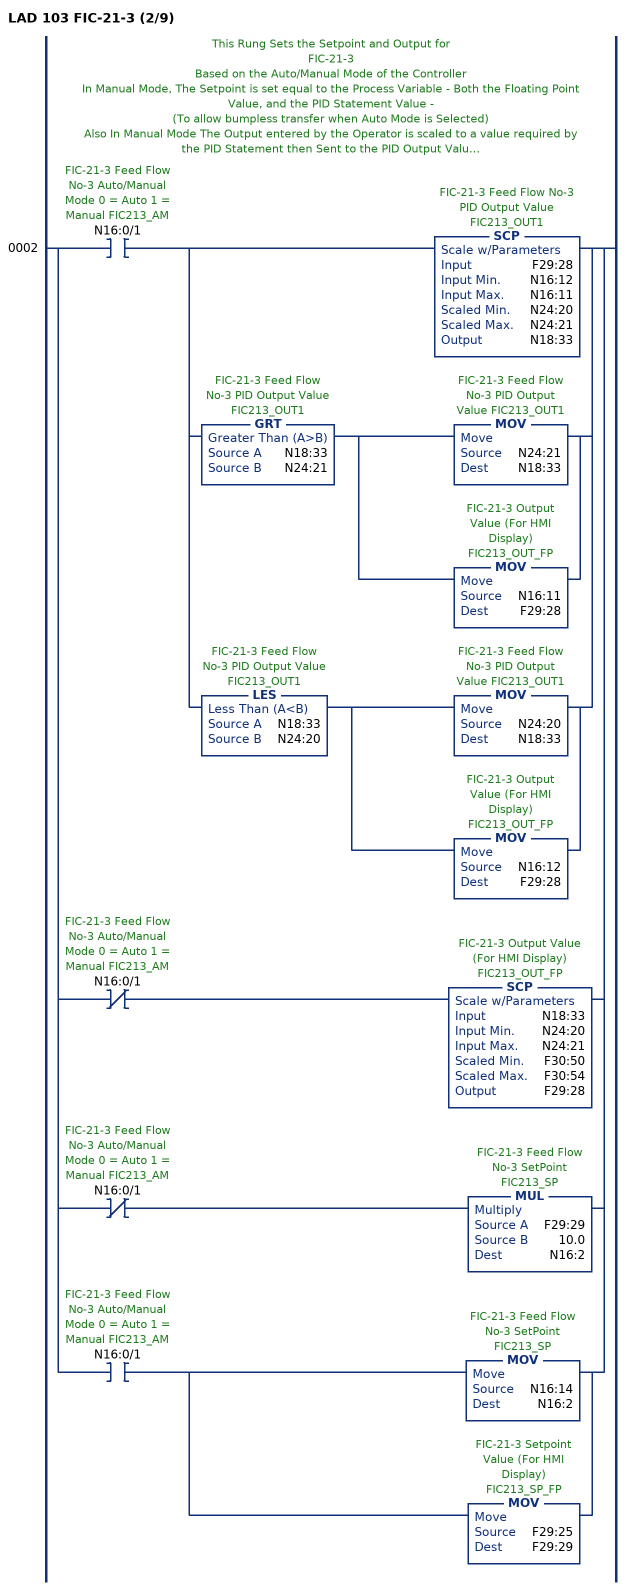
% Rung: 2 %
% This Rung Sets the Setpoint and Output for
% FIC-21-3
% Based on the Auto/Manual Mode of the Controller
% In Manual Mode, The Setpoint is set equal to the Process Variable - Both the Floating Point Value, and the PID Statement Value -
% (To allow bumpless transfer when Auto Mode is Selected)
% Also In Manual Mode The Output entered by the Operator is scaled to a value required by the PID Statement then Sent to the PID Output Value
% 
% In Auto Mode, The Setpoint is Entered by the Operator from Any HMI terminal, Multiplied by 10, and placed in the PID Statement's Setpoint Location
% Also In Auto Mode, the Output (used by the Operator) is set equal to the actual value of the pID statement
% (To allow bumpless transfer when Manual Mode is Selected) %
SOR BST XIC N16:0/1 BST SCP F29:28 N16:12 N16:11 N24:20 N24:21 N18:33 NXB GRT N18:33 N24:21 BST MOV N24:21 N18:33 NXB MOV N16:11 F29:28 BND NXB LES N18:33 N24:20 BST MOV N24:20 N18:33 NXB MOV N16:12 F29:28 BND BND NXB XIO N16:0/1 SCP N18:33 N24:20 N24:21 F30:50 F30:54 F29:28 NXB XIO N16:0/1 MUL F29:29 10.0 N16:2 NXB XIC N16:0/1 BST MOV N16:14 N16:2 NXB MOV F29:25 F29:29 BND BND EOR
%   N16:0/1  FIC213_AM  "FIC-21-3 Feed Flow No-3 Auto/Manual Mode 0 = Auto 1 = Manual" %
%   F29:28  FIC213_OUT_FP  "FIC-21-3 Output Value (For HMI Display)" %
%   N16:12  FIC213_OMIN  "FIC-21-3 Feed Flow No-3 Output Minimum" %
%   N16:11  FIC213_OMAX  "FIC-21-3 Feed Flow No-3 Output Maximum" %
%   N24:20  PID_MIN  "PID Statement Minimum Value" %
%   N24:21  PID_MAX  "PID Statement Maximum Value" %
%   N18:33  FIC213_OUT1  "FIC-21-3 Feed Flow No-3 PID Output Value" %
%   F30:50  SIC213_MIN  "SIC-21-3 PU-21-3 Feed Pump No-3 Speed 0% Value (For HMI Display)" %
%   F30:54  SIC213_MAX  "SIC-21-3 PU-21-3 Feed Pump No-3 Freq at 100% Value (For HMI Display)" %
%   F29:29  FIC213_SP_FP  "FIC-21-3 Setpoint Value (For HMI Display)" %
%   N16:2  FIC213_SP  "FIC-21-3 Feed Flow No-3 SetPoint" %
%   N16:14  FIC213_PV  "FIC-21-3 Feed Flow No-3 Scaled Process Variable" %
%   F29:25  FIC213_PV_FP  "FIC-21-3 PV Value (For HMI Display)" %

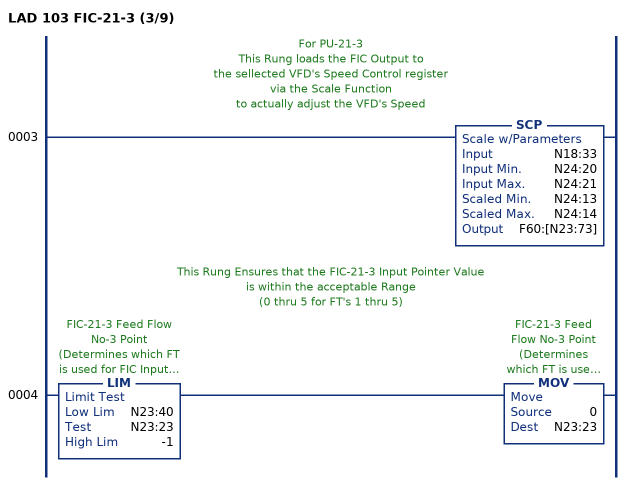
% Rung: 3 %
% For PU-21-3
% This Rung loads the FIC Output to
% the sellected VFD's Speed Control register
% via the Scale Function
% to actually adjust the VFD's Speed %
SOR SCP N18:33 N24:20 N24:21 N24:13 N24:14 F60:[N23:73] EOR
%   N18:33  FIC213_OUT1  "FIC-21-3 Feed Flow No-3 PID Output Value" %
%   N24:20  PID_MIN  "PID Statement Minimum Value" %
%   N24:21  PID_MAX  "PID Statement Maximum Value" %
%   N24:13  AO_MIN_OE4  "Analog Output Minimum Value Generates 4 mA DC (To OE4 AO Module)" %
%   N24:14  AO_MAX_OE4  "Analog Output Maximum Value Generates 20 mA DC (To OE4 AO Module)" %
%   N23:73  FIC213_OUT_PTR  "FIC-21-3 Feed Flow No-3 Output Pointer Determines which VFD is controled by FIC" %
% Rung: 4 %
% This Rung Ensures that the FIC-21-3 Input Pointer Value
% is within the acceptable Range
% (0 thru 5 for FT's 1 thru 5) %
SOR LIM N23:40 N23:23 -1 MOV 0 N23:23 EOR
%   N23:40  MAX_FT_ALLOWED_1  "Maximum Number of FTs Available Plus 1" %
%   N23:23  FIC213_IN_PTR  "FIC-21-3 Feed Flow No-3 Point (Determines which FT is used for FIC Input)" %

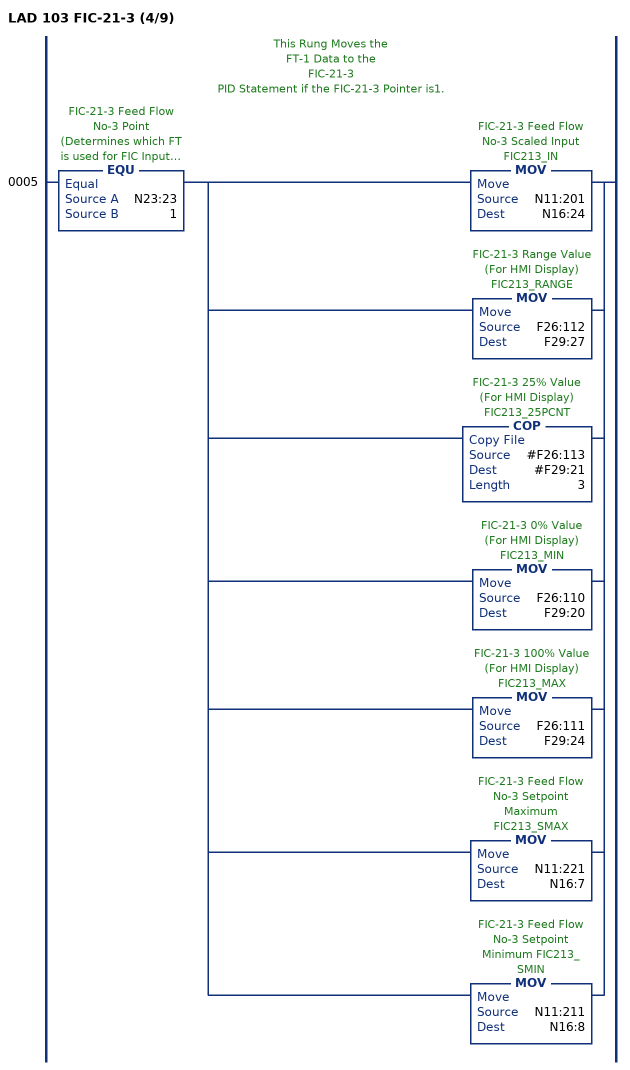
% Rung: 5 %
% This Rung Moves the
% FT-1 Data to the
% FIC-21-3
% PID Statement if the FIC-21-3 Pointer is1. %
SOR EQU N23:23 1 BST MOV N11:201 N16:24 NXB MOV F26:112 F29:27 NXB COP #F26:113 #F29:21 3 NXB MOV F26:110 F29:20 NXB MOV F26:111 F29:24 NXB MOV N11:221 N16:7 NXB MOV N11:211 N16:8 BND EOR
%   N23:23  FIC213_IN_PTR  "FIC-21-3 Feed Flow No-3 Point (Determines which FT is used for FIC Input)" %
%   N11:201  FT01_PID_IN  "FT-1 Flow Transmitter No-1 PID Statement Input Value" %
%   N16:24  FIC213_IN  "FIC-21-3 Feed Flow No-3 Scaled Input" %
%   F26:112  FT01_RANGE  "FT-1 Range Value (Max-Min)" %
%   F29:27  FIC213_RANGE  "FIC-21-3 Range Value (For HMI Display)" %
%   F26:113  FT01_25PCNT_VALUE  "FT-1 25% Range Value For HMI Display" %
%   F29:21  FIC213_25PCNT  "FIC-21-3 25% Value (For HMI Display)" %
%   F26:110  FT01_MIN  "FT-1 Minimum Value" %
%   F29:20  FIC213_MIN  "FIC-21-3 0% Value (For HMI Display)" %
%   F26:111  FT01_MAX  "FT-1 Maximum Value" %
%   F29:24  FIC213_MAX  "FIC-21-3 100% Value (For HMI Display)" %
%   N11:221  FT01_PID_MAX  "FT-1 Flow Transmitter No-1 PID Statement Maximum Input Value" %
%   N16:7  FIC213_SMAX  "FIC-21-3 Feed Flow No-3 Setpoint Maximum" %
%   N11:211  FT01_PID_MIN  "FT-1 Flow Transmitter No-1 PID Statement Minimum Input Value" %
%   N16:8  FIC213_SMIN  "FIC-21-3 Feed Flow No-3 Setpoint Minimum" %

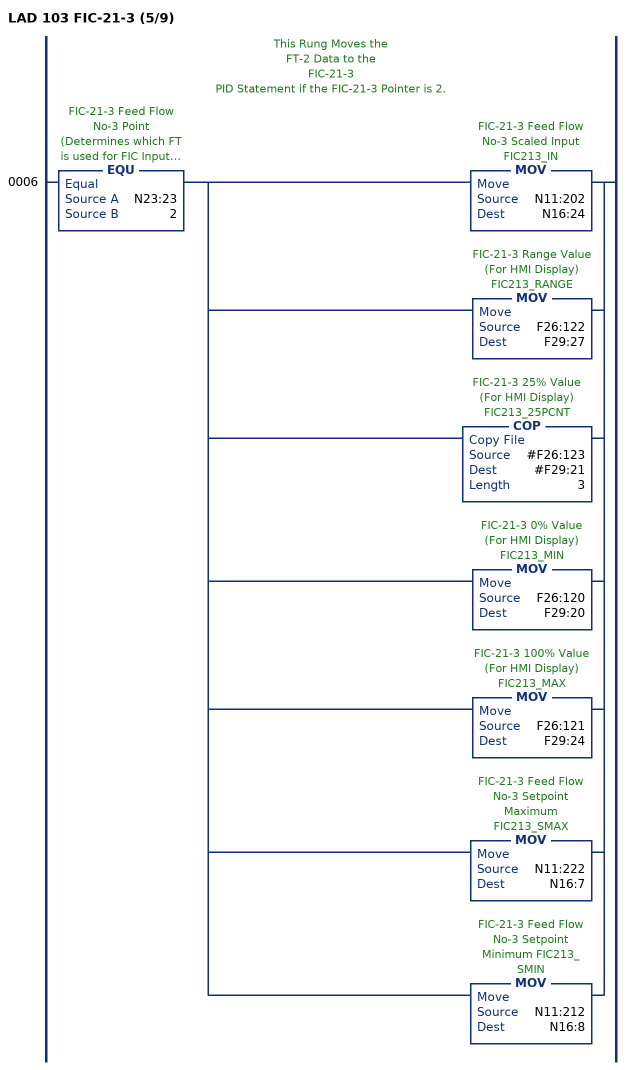
% Rung: 6 %
% This Rung Moves the
% FT-2 Data to the
% FIC-21-3
% PID Statement if the FIC-21-3 Pointer is 2. %
SOR EQU N23:23 2 BST MOV N11:202 N16:24 NXB MOV F26:122 F29:27 NXB COP #F26:123 #F29:21 3 NXB MOV F26:120 F29:20 NXB MOV F26:121 F29:24 NXB MOV N11:222 N16:7 NXB MOV N11:212 N16:8 BND EOR
%   N23:23  FIC213_IN_PTR  "FIC-21-3 Feed Flow No-3 Point (Determines which FT is used for FIC Input)" %
%   N11:202  FT02_PID_IN  "FT-2 Flow Transmitter No-2 PID Statement Input Value" %
%   N16:24  FIC213_IN  "FIC-21-3 Feed Flow No-3 Scaled Input" %
%   F26:122  FT02_RANGE  "FT-2 Range Value (Max-Min)" %
%   F29:27  FIC213_RANGE  "FIC-21-3 Range Value (For HMI Display)" %
%   F26:123  FT02_25PCNT_VALUE  "FT-2 25% Range Value For HMI Display" %
%   F29:21  FIC213_25PCNT  "FIC-21-3 25% Value (For HMI Display)" %
%   F26:120  FT02_MIN  "FT-2 Minimum Value" %
%   F29:20  FIC213_MIN  "FIC-21-3 0% Value (For HMI Display)" %
%   F26:121  FT02_MAX  "FT-2 Maximum Value" %
%   F29:24  FIC213_MAX  "FIC-21-3 100% Value (For HMI Display)" %
%   N11:222  FT02_PID_MAX  "FT-2 Flow Transmitter No-2 PID Statement Maximum Input Value" %
%   N16:7  FIC213_SMAX  "FIC-21-3 Feed Flow No-3 Setpoint Maximum" %
%   N11:212  FT02_PID_MIN  "FT-2 Flow Transmitter No-2 PID Statement Minimum Input Value" %
%   N16:8  FIC213_SMIN  "FIC-21-3 Feed Flow No-3 Setpoint Minimum" %

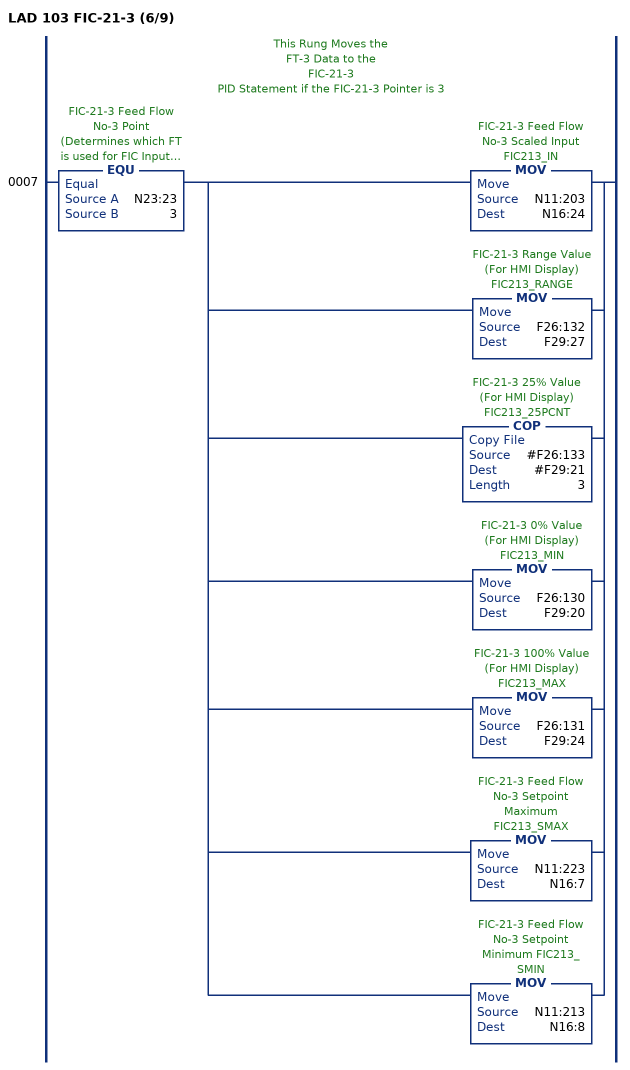
% Rung: 7 %
% This Rung Moves the
% FT-3 Data to the
% FIC-21-3
% PID Statement if the FIC-21-3 Pointer is 3 %
SOR EQU N23:23 3 BST MOV N11:203 N16:24 NXB MOV F26:132 F29:27 NXB COP #F26:133 #F29:21 3 NXB MOV F26:130 F29:20 NXB MOV F26:131 F29:24 NXB MOV N11:223 N16:7 NXB MOV N11:213 N16:8 BND EOR
%   N23:23  FIC213_IN_PTR  "FIC-21-3 Feed Flow No-3 Point (Determines which FT is used for FIC Input)" %
%   N11:203  FT03_PID_IN  "FT-3 Flow Transmitter No-3 PID Statement Input Value" %
%   N16:24  FIC213_IN  "FIC-21-3 Feed Flow No-3 Scaled Input" %
%   F26:132  FT03_RANGE  "FT-3 Range Value (Max-Min)" %
%   F29:27  FIC213_RANGE  "FIC-21-3 Range Value (For HMI Display)" %
%   F26:133  FT03_25PCNT_VALUE  "FT-3 25% Range Value For HMI Display" %
%   F29:21  FIC213_25PCNT  "FIC-21-3 25% Value (For HMI Display)" %
%   F26:130  FT03_MIN  "FT-3 Minimum Value" %
%   F29:20  FIC213_MIN  "FIC-21-3 0% Value (For HMI Display)" %
%   F26:131  FT03_MAX  "FT-3 Maximum Value" %
%   F29:24  FIC213_MAX  "FIC-21-3 100% Value (For HMI Display)" %
%   N11:223  FT03_PID_MAX  "FT-3 Flow Transmitter No-3 PID Statement Maximum Input Value" %
%   N16:7  FIC213_SMAX  "FIC-21-3 Feed Flow No-3 Setpoint Maximum" %
%   N11:213  FT03_PID_MIN  "FT-3 Flow Transmitter No-3 PID Statement Minimum Input Value" %
%   N16:8  FIC213_SMIN  "FIC-21-3 Feed Flow No-3 Setpoint Minimum" %

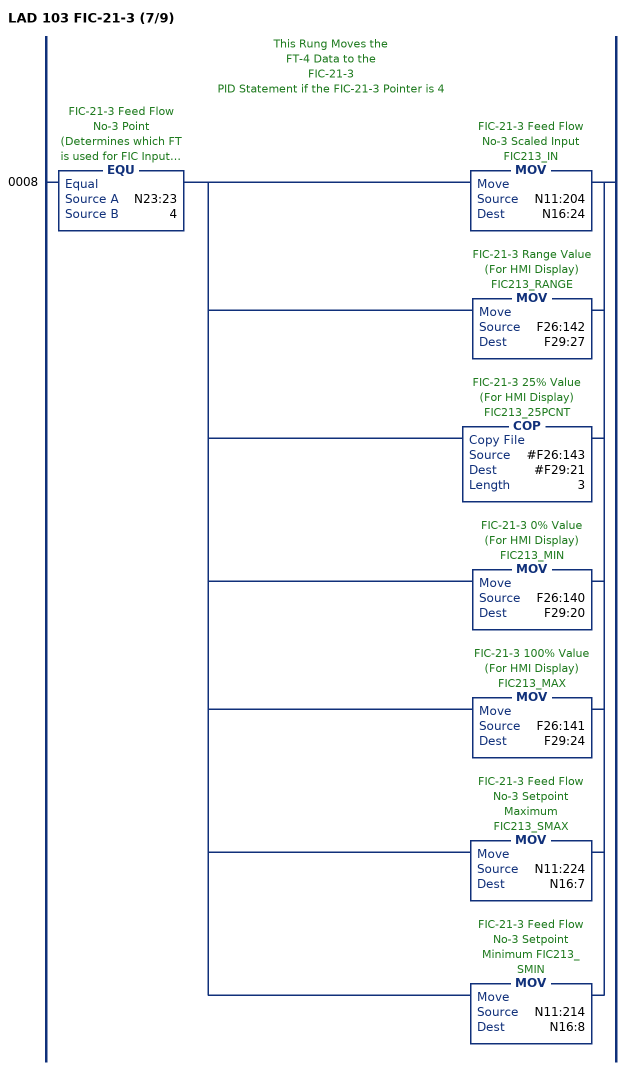
% Rung: 8 %
% This Rung Moves the
% FT-4 Data to the
% FIC-21-3
% PID Statement if the FIC-21-3 Pointer is 4 %
SOR EQU N23:23 4 BST MOV N11:204 N16:24 NXB MOV F26:142 F29:27 NXB COP #F26:143 #F29:21 3 NXB MOV F26:140 F29:20 NXB MOV F26:141 F29:24 NXB MOV N11:224 N16:7 NXB MOV N11:214 N16:8 BND EOR
%   N23:23  FIC213_IN_PTR  "FIC-21-3 Feed Flow No-3 Point (Determines which FT is used for FIC Input)" %
%   N11:204  FT04_PID_IN  "FT-4 Flow Transmitter No-4 PID Statement Input Value" %
%   N16:24  FIC213_IN  "FIC-21-3 Feed Flow No-3 Scaled Input" %
%   F26:142  FT04_RANGE  "FT-4 Range Value (Max-Min)" %
%   F29:27  FIC213_RANGE  "FIC-21-3 Range Value (For HMI Display)" %
%   F26:143  FT04_25PCNT_VALUE  "FT-4 25% Range Value For HMI Display" %
%   F29:21  FIC213_25PCNT  "FIC-21-3 25% Value (For HMI Display)" %
%   F26:140  FT04_MIN  "FT-4 Minimum Value" %
%   F29:20  FIC213_MIN  "FIC-21-3 0% Value (For HMI Display)" %
%   F26:141  FT04_MAX  "FT-4 Maximum Value" %
%   F29:24  FIC213_MAX  "FIC-21-3 100% Value (For HMI Display)" %
%   N11:224  FT04_PID_MAX  "FT-4 Flow Transmitter No-4 PID Statement Maximum Input Value" %
%   N16:7  FIC213_SMAX  "FIC-21-3 Feed Flow No-3 Setpoint Maximum" %
%   N11:214  FT04_PID_MIN  "FT-4 Flow Transmitter No-4 PID Statement Minimum Input Value" %
%   N16:8  FIC213_SMIN  "FIC-21-3 Feed Flow No-3 Setpoint Minimum" %

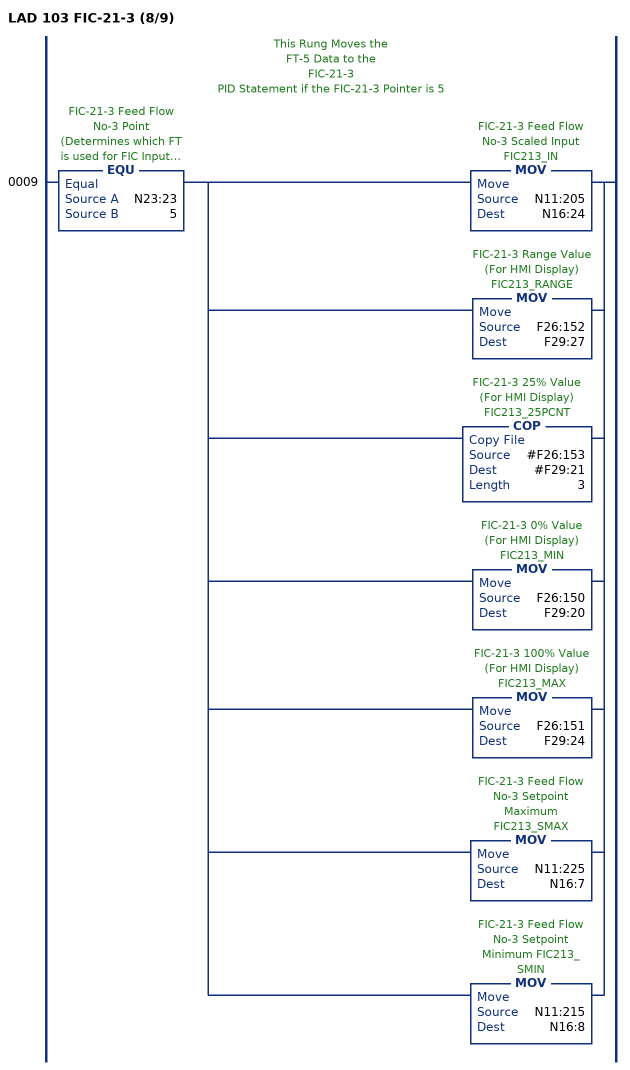
% Rung: 9 %
% This Rung Moves the
% FT-5 Data to the
% FIC-21-3
%  PID Statement if the FIC-21-3 Pointer is 5 %
SOR EQU N23:23 5 BST MOV N11:205 N16:24 NXB MOV F26:152 F29:27 NXB COP #F26:153 #F29:21 3 NXB MOV F26:150 F29:20 NXB MOV F26:151 F29:24 NXB MOV N11:225 N16:7 NXB MOV N11:215 N16:8 BND EOR
%   N23:23  FIC213_IN_PTR  "FIC-21-3 Feed Flow No-3 Point (Determines which FT is used for FIC Input)" %
%   N11:205  FT05_PID_IN  "FT-5 Flow Transmitter No-5 PID Statement Input Value" %
%   N16:24  FIC213_IN  "FIC-21-3 Feed Flow No-3 Scaled Input" %
%   F26:152  FT05_RANGE  "FT-5 Range Value (Max-Min)" %
%   F29:27  FIC213_RANGE  "FIC-21-3 Range Value (For HMI Display)" %
%   F26:153  FT05_25PCNT_VALUE  "FT-5 25% Range Value For HMI Display" %
%   F29:21  FIC213_25PCNT  "FIC-21-3 25% Value (For HMI Display)" %
%   F26:150  FT05_MIN  "FT-5 Minimum Value" %
%   F29:20  FIC213_MIN  "FIC-21-3 0% Value (For HMI Display)" %
%   F26:151  FT05_MAX  "FT-5 Maximum Value" %
%   F29:24  FIC213_MAX  "FIC-21-3 100% Value (For HMI Display)" %
%   N11:225  FT05_PID_MAX  "FT-5 Flow Transmitter No-5 PID Statement Maximum Input Value" %
%   N16:7  FIC213_SMAX  "FIC-21-3 Feed Flow No-3 Setpoint Maximum" %
%   N11:215  FT05_PID_MIN  "FT-5 Flow Transmitter No-5 PID Statement Minimum Input Value" %
%   N16:8  FIC213_SMIN  "FIC-21-3 Feed Flow No-3 Setpoint Minimum" %

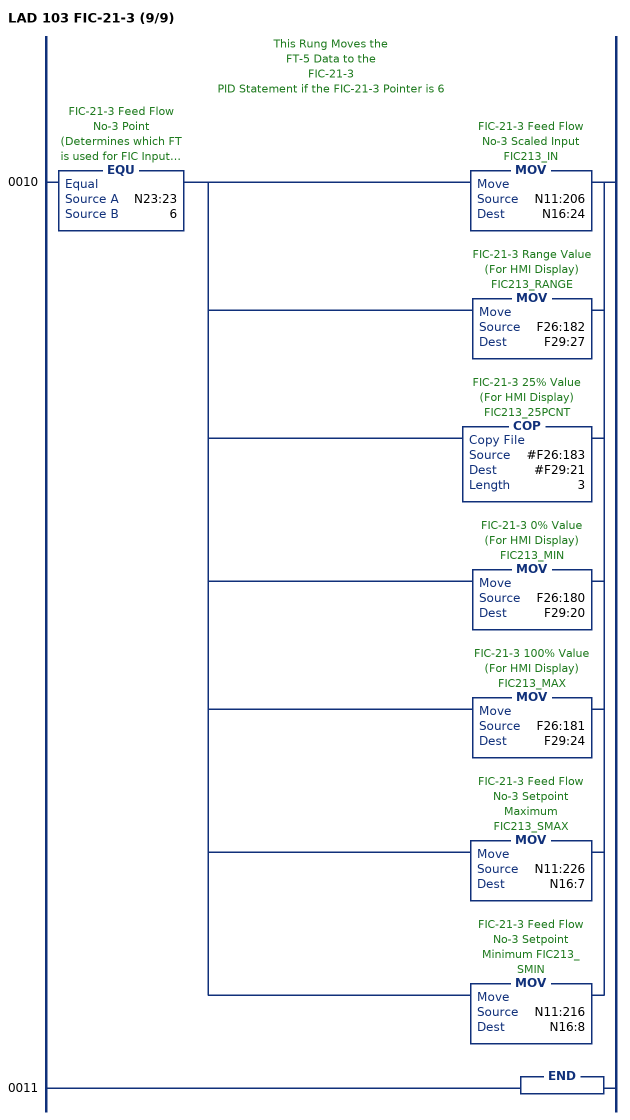
% Rung: 10 %
% This Rung Moves the
% FT-5 Data to the
% FIC-21-3
%  PID Statement if the FIC-21-3 Pointer is 6 %
SOR EQU N23:23 6 BST MOV N11:206 N16:24 NXB MOV F26:182 F29:27 NXB COP #F26:183 #F29:21 3 NXB MOV F26:180 F29:20 NXB MOV F26:181 F29:24 NXB MOV N11:226 N16:7 NXB MOV N11:216 N16:8 BND EOR
%   N23:23  FIC213_IN_PTR  "FIC-21-3 Feed Flow No-3 Point (Determines which FT is used for FIC Input)" %
%   N11:206  FT06_PID_IN  "FT-6 Flow Transmitter No-6 PID Statement Input Value" %
%   N16:24  FIC213_IN  "FIC-21-3 Feed Flow No-3 Scaled Input" %
%   F26:182  FT06_RANGE  "FT-6 Range Value (Max-Min)" %
%   F29:27  FIC213_RANGE  "FIC-21-3 Range Value (For HMI Display)" %
%   F26:183  FT06_25PCNT_VALUE  "FT-6 25% Range Value For HMI Display" %
%   F29:21  FIC213_25PCNT  "FIC-21-3 25% Value (For HMI Display)" %
%   F26:180  FT06_MIN  "FT-6 Minimum Value" %
%   F29:20  FIC213_MIN  "FIC-21-3 0% Value (For HMI Display)" %
%   F26:181  FT06_MAX  "FT-6 Maximum Value" %
%   F29:24  FIC213_MAX  "FIC-21-3 100% Value (For HMI Display)" %
%   N11:226  FT06_PID_MAX  "FT-6 Flow Transmitter No-6 PID Statement Maximum Input Value" %
%   N16:7  FIC213_SMAX  "FIC-21-3 Feed Flow No-3 Setpoint Maximum" %
%   N11:216  FT06_PID_MIN  "FT-6 Flow Transmitter No-6 PID Statement Minimum Input Value" %
%   N16:8  FIC213_SMIN  "FIC-21-3 Feed Flow No-3 Setpoint Minimum" %
% Rung: 11 %
SOR END EOR

LADDER 104 "FIC-21-4"    % Feed Flow No-4 PID Controls %
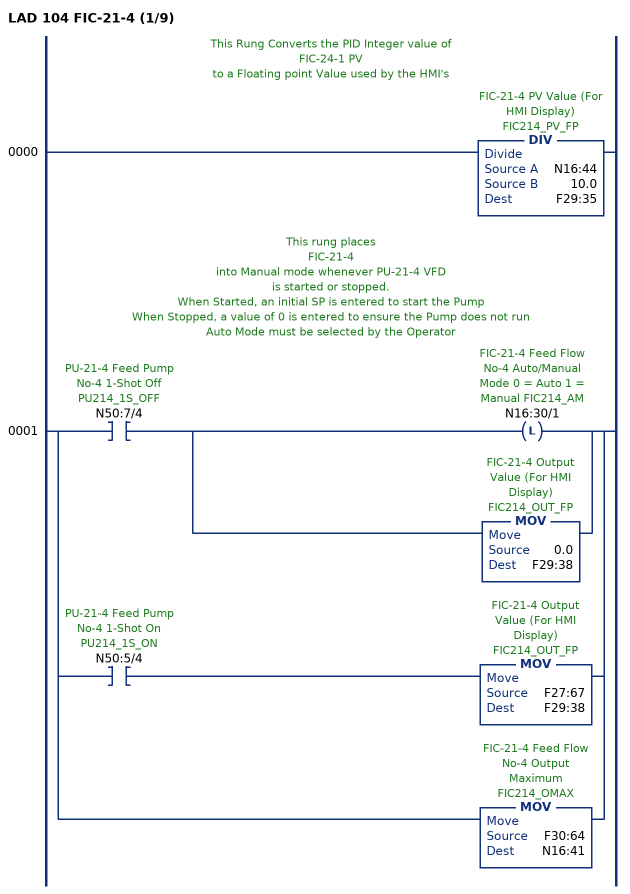
% Rung: 0 %
% This Rung Converts the PID Integer value of
% FIC-24-1 PV
% to a Floating point Value used by the HMI's %
SOR DIV N16:44 10.0 F29:35 EOR
%   N16:44  FIC214_PV  "FIC-21-4 Feed Flow No-4 Scaled Process Variable" %
%   F29:35  FIC214_PV_FP  "FIC-21-4 PV Value (For HMI Display)" %
% Rung: 1 %
% This rung places
% FIC-21-4
% into Manual mode whenever PU-21-4 VFD
% is started or stopped.
% When Started, an initial SP is entered to start the Pump
% When Stopped, a value of 0 is entered to ensure the Pump does not run
% Auto Mode must be selected by the Operator %
SOR BST XIC N50:7/4 BST OTL N16:30/1 NXB MOV 0.0 F29:38 BND NXB XIC N50:5/4 MOV F27:67 F29:38 NXB MOV F30:64 N16:41 BND EOR
%   N50:7/4  PU214_1S_OFF  "PU-21-4 Feed Pump No-4 1-Shot Off" %
%   N16:30/1  FIC214_AM  "FIC-21-4 Feed Flow No-4 Auto/Manual Mode 0 = Auto 1 = Manual" %
%   F29:38  FIC214_OUT_FP  "FIC-21-4 Output Value (For HMI Display)" %
%   N50:5/4  PU214_1S_ON  "PU-21-4 Feed Pump No-4 1-Shot On" %
%   F27:67  SIC214_INIT_SP  "SIC-21-4 Initial Speed Setpoint (Hz)" %
%   F30:64  SIC214_MAX  "SIC-21-4 PU-21-4 Feed Pump No-4 Freq at 100% Value (For HMI Display)" %
%   N16:41  FIC214_OMAX  "FIC-21-4 Feed Flow No-4 Output Maximum" %

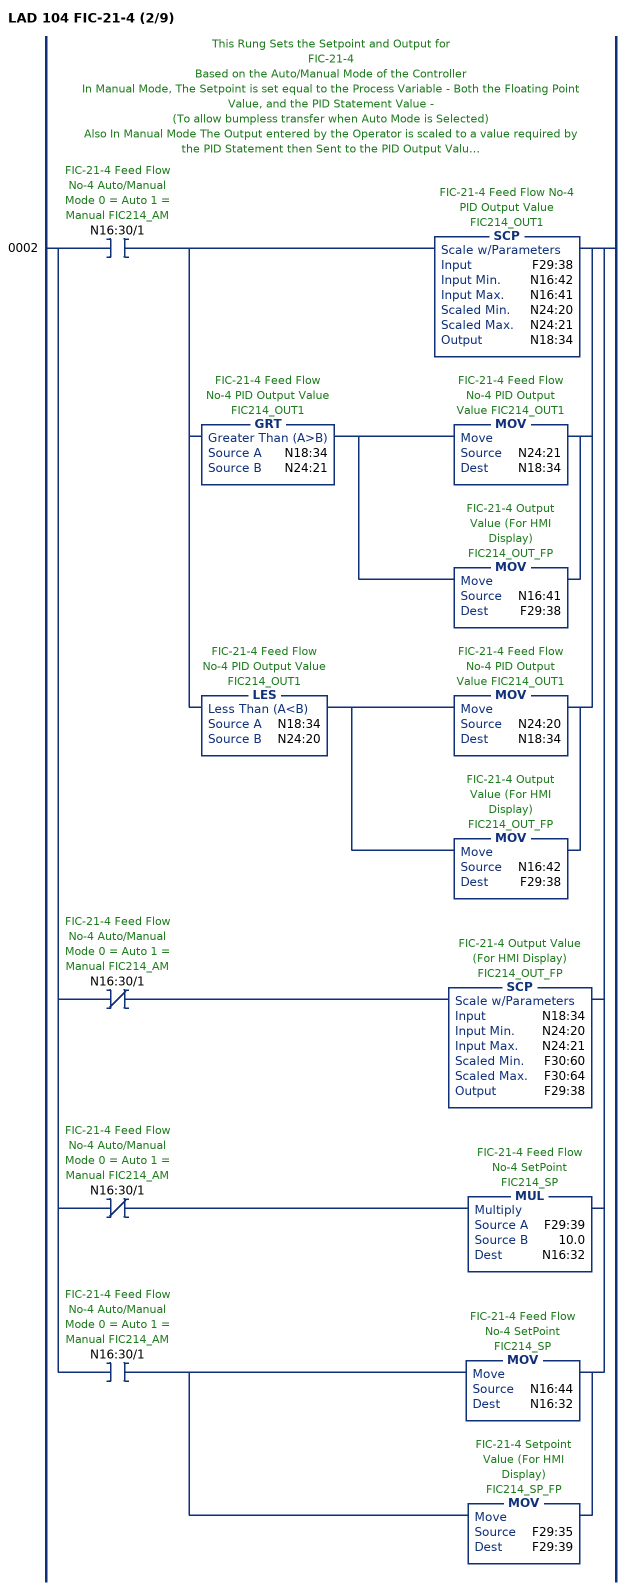
% Rung: 2 %
% This Rung Sets the Setpoint and Output for
% FIC-21-4
% Based on the Auto/Manual Mode of the Controller
% In Manual Mode, The Setpoint is set equal to the Process Variable - Both the Floating Point Value, and the PID Statement Value -
% (To allow bumpless transfer when Auto Mode is Selected)
% Also In Manual Mode The Output entered by the Operator is scaled to a value required by the PID Statement then Sent to the PID Output Value
% 
% In Auto Mode, The Setpoint is Entered by the Operator from Any HMI terminal, Multiplied by 10, and placed in the PID Statement's Setpoint Location
% Also In Auto Mode, the Output (used by the Operator) is set equal to the actual value of the pID statement
% (To allow bumpless transfer when Manual Mode is Selected) %
SOR BST XIC N16:30/1 BST SCP F29:38 N16:42 N16:41 N24:20 N24:21 N18:34 NXB GRT N18:34 N24:21 BST MOV N24:21 N18:34 NXB MOV N16:41 F29:38 BND NXB LES N18:34 N24:20 BST MOV N24:20 N18:34 NXB MOV N16:42 F29:38 BND BND NXB XIO N16:30/1 SCP N18:34 N24:20 N24:21 F30:60 F30:64 F29:38 NXB XIO N16:30/1 MUL F29:39 10.0 N16:32 NXB XIC N16:30/1 BST MOV N16:44 N16:32 NXB MOV F29:35 F29:39 BND BND EOR
%   N16:30/1  FIC214_AM  "FIC-21-4 Feed Flow No-4 Auto/Manual Mode 0 = Auto 1 = Manual" %
%   F29:38  FIC214_OUT_FP  "FIC-21-4 Output Value (For HMI Display)" %
%   N16:42  FIC214_OMIN  "FIC-21-4 Feed Flow No-4 Output Minimum" %
%   N16:41  FIC214_OMAX  "FIC-21-4 Feed Flow No-4 Output Maximum" %
%   N24:20  PID_MIN  "PID Statement Minimum Value" %
%   N24:21  PID_MAX  "PID Statement Maximum Value" %
%   N18:34  FIC214_OUT1  "FIC-21-4 Feed Flow No-4 PID Output Value" %
%   F30:60  SIC214_MIN  "SIC-21-4 PU-21-4 Feed Pump No-4 Speed 0% Value (For HMI Display)" %
%   F30:64  SIC214_MAX  "SIC-21-4 PU-21-4 Feed Pump No-4 Freq at 100% Value (For HMI Display)" %
%   F29:39  FIC214_SP_FP  "FIC-21-4 Setpoint Value (For HMI Display)" %
%   N16:32  FIC214_SP  "FIC-21-4 Feed Flow No-4 SetPoint" %
%   N16:44  FIC214_PV  "FIC-21-4 Feed Flow No-4 Scaled Process Variable" %
%   F29:35  FIC214_PV_FP  "FIC-21-4 PV Value (For HMI Display)" %

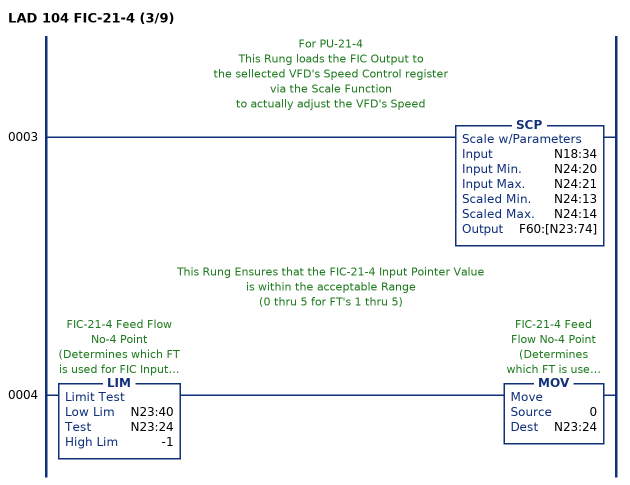
% Rung: 3 %
% For PU-21-4
% This Rung loads the FIC Output to
% the sellected VFD's Speed Control register
% via the Scale Function
% to actually adjust the VFD's Speed %
SOR SCP N18:34 N24:20 N24:21 N24:13 N24:14 F60:[N23:74] EOR
%   N18:34  FIC214_OUT1  "FIC-21-4 Feed Flow No-4 PID Output Value" %
%   N24:20  PID_MIN  "PID Statement Minimum Value" %
%   N24:21  PID_MAX  "PID Statement Maximum Value" %
%   N24:13  AO_MIN_OE4  "Analog Output Minimum Value Generates 4 mA DC (To OE4 AO Module)" %
%   N24:14  AO_MAX_OE4  "Analog Output Maximum Value Generates 20 mA DC (To OE4 AO Module)" %
%   N23:74  FIC214_OUT_PTR  "FIC-21-4 Feed Flow No-4 Output Pointer Determines which VFD is controled by FIC" %
% Rung: 4 %
% This Rung Ensures that the FIC-21-4 Input Pointer Value
% is within the acceptable Range
% (0 thru 5 for FT's 1 thru 5) %
SOR LIM N23:40 N23:24 -1 MOV 0 N23:24 EOR
%   N23:40  MAX_FT_ALLOWED_1  "Maximum Number of FTs Available Plus 1" %
%   N23:24  FIC214_IN_PTR  "FIC-21-4 Feed Flow No-4 Point (Determines which FT is used for FIC Input)" %

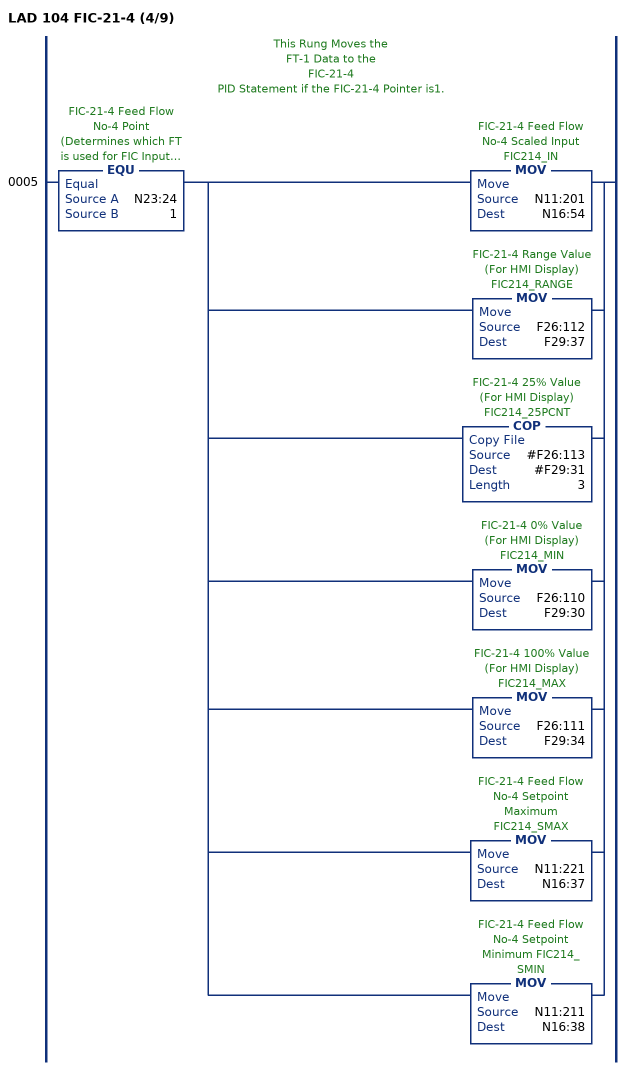
% Rung: 5 %
% This Rung Moves the
% FT-1 Data to the
% FIC-21-4
% PID Statement if the FIC-21-4 Pointer is1. %
SOR EQU N23:24 1 BST MOV N11:201 N16:54 NXB MOV F26:112 F29:37 NXB COP #F26:113 #F29:31 3 NXB MOV F26:110 F29:30 NXB MOV F26:111 F29:34 NXB MOV N11:221 N16:37 NXB MOV N11:211 N16:38 BND EOR
%   N23:24  FIC214_IN_PTR  "FIC-21-4 Feed Flow No-4 Point (Determines which FT is used for FIC Input)" %
%   N11:201  FT01_PID_IN  "FT-1 Flow Transmitter No-1 PID Statement Input Value" %
%   N16:54  FIC214_IN  "FIC-21-4 Feed Flow No-4 Scaled Input" %
%   F26:112  FT01_RANGE  "FT-1 Range Value (Max-Min)" %
%   F29:37  FIC214_RANGE  "FIC-21-4 Range Value (For HMI Display)" %
%   F26:113  FT01_25PCNT_VALUE  "FT-1 25% Range Value For HMI Display" %
%   F29:31  FIC214_25PCNT  "FIC-21-4 25% Value (For HMI Display)" %
%   F26:110  FT01_MIN  "FT-1 Minimum Value" %
%   F29:30  FIC214_MIN  "FIC-21-4 0% Value (For HMI Display)" %
%   F26:111  FT01_MAX  "FT-1 Maximum Value" %
%   F29:34  FIC214_MAX  "FIC-21-4 100% Value (For HMI Display)" %
%   N11:221  FT01_PID_MAX  "FT-1 Flow Transmitter No-1 PID Statement Maximum Input Value" %
%   N16:37  FIC214_SMAX  "FIC-21-4 Feed Flow No-4 Setpoint Maximum" %
%   N11:211  FT01_PID_MIN  "FT-1 Flow Transmitter No-1 PID Statement Minimum Input Value" %
%   N16:38  FIC214_SMIN  "FIC-21-4 Feed Flow No-4 Setpoint Minimum" %

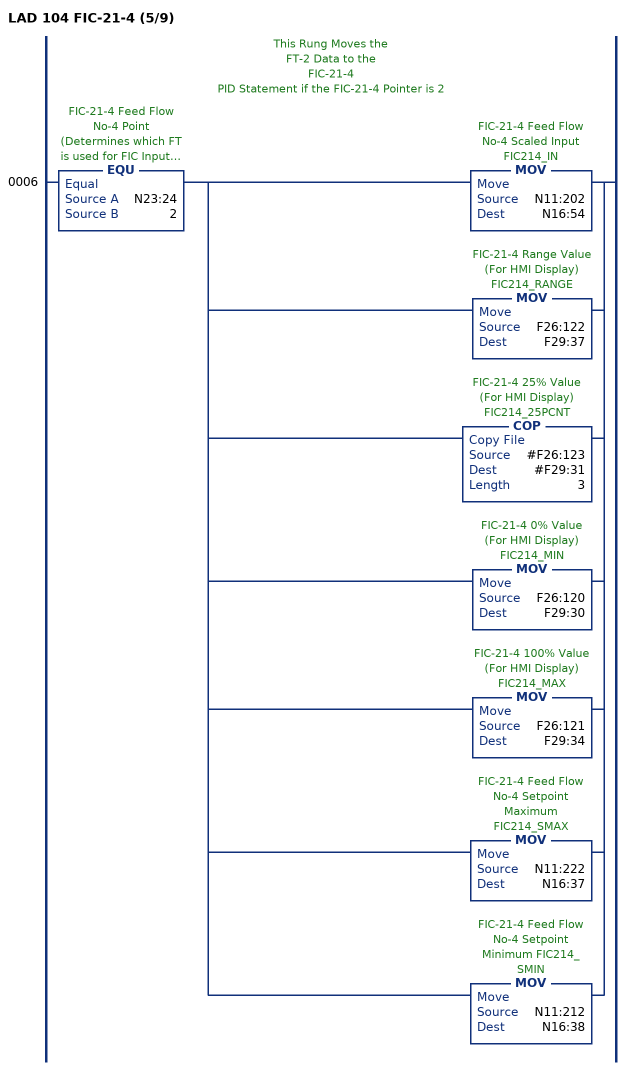
% Rung: 6 %
% This Rung Moves the
% FT-2 Data to the
% FIC-21-4
% PID Statement if the FIC-21-4 Pointer is 2 %
SOR EQU N23:24 2 BST MOV N11:202 N16:54 NXB MOV F26:122 F29:37 NXB COP #F26:123 #F29:31 3 NXB MOV F26:120 F29:30 NXB MOV F26:121 F29:34 NXB MOV N11:222 N16:37 NXB MOV N11:212 N16:38 BND EOR
%   N23:24  FIC214_IN_PTR  "FIC-21-4 Feed Flow No-4 Point (Determines which FT is used for FIC Input)" %
%   N11:202  FT02_PID_IN  "FT-2 Flow Transmitter No-2 PID Statement Input Value" %
%   N16:54  FIC214_IN  "FIC-21-4 Feed Flow No-4 Scaled Input" %
%   F26:122  FT02_RANGE  "FT-2 Range Value (Max-Min)" %
%   F29:37  FIC214_RANGE  "FIC-21-4 Range Value (For HMI Display)" %
%   F26:123  FT02_25PCNT_VALUE  "FT-2 25% Range Value For HMI Display" %
%   F29:31  FIC214_25PCNT  "FIC-21-4 25% Value (For HMI Display)" %
%   F26:120  FT02_MIN  "FT-2 Minimum Value" %
%   F29:30  FIC214_MIN  "FIC-21-4 0% Value (For HMI Display)" %
%   F26:121  FT02_MAX  "FT-2 Maximum Value" %
%   F29:34  FIC214_MAX  "FIC-21-4 100% Value (For HMI Display)" %
%   N11:222  FT02_PID_MAX  "FT-2 Flow Transmitter No-2 PID Statement Maximum Input Value" %
%   N16:37  FIC214_SMAX  "FIC-21-4 Feed Flow No-4 Setpoint Maximum" %
%   N11:212  FT02_PID_MIN  "FT-2 Flow Transmitter No-2 PID Statement Minimum Input Value" %
%   N16:38  FIC214_SMIN  "FIC-21-4 Feed Flow No-4 Setpoint Minimum" %

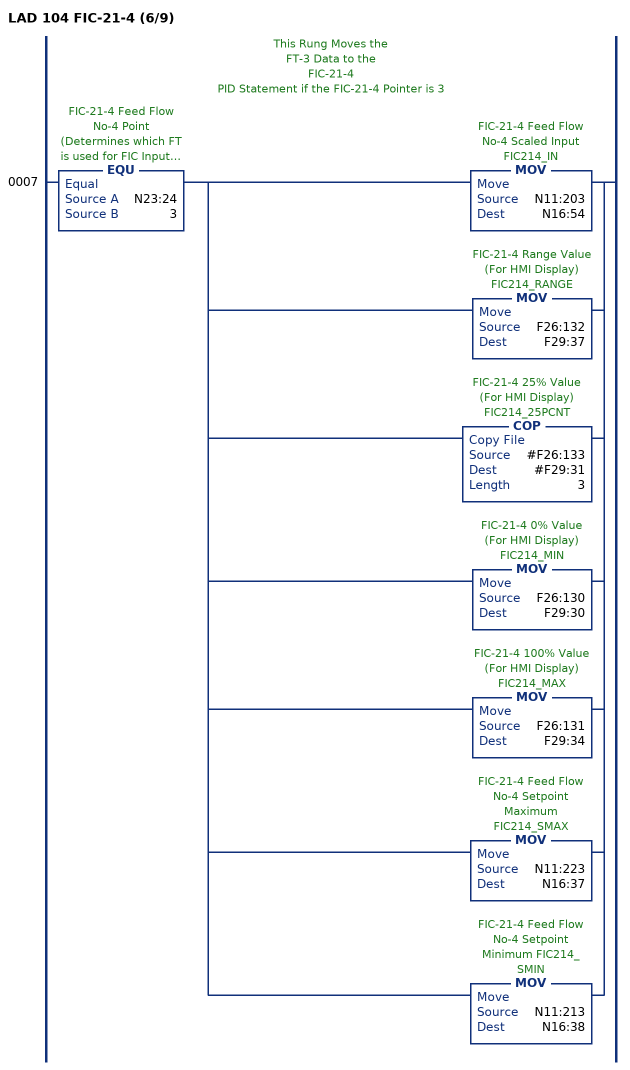
% Rung: 7 %
% This Rung Moves the
% FT-3 Data to the
% FIC-21-4
% PID Statement if the FIC-21-4 Pointer is 3 %
SOR EQU N23:24 3 BST MOV N11:203 N16:54 NXB MOV F26:132 F29:37 NXB COP #F26:133 #F29:31 3 NXB MOV F26:130 F29:30 NXB MOV F26:131 F29:34 NXB MOV N11:223 N16:37 NXB MOV N11:213 N16:38 BND EOR
%   N23:24  FIC214_IN_PTR  "FIC-21-4 Feed Flow No-4 Point (Determines which FT is used for FIC Input)" %
%   N11:203  FT03_PID_IN  "FT-3 Flow Transmitter No-3 PID Statement Input Value" %
%   N16:54  FIC214_IN  "FIC-21-4 Feed Flow No-4 Scaled Input" %
%   F26:132  FT03_RANGE  "FT-3 Range Value (Max-Min)" %
%   F29:37  FIC214_RANGE  "FIC-21-4 Range Value (For HMI Display)" %
%   F26:133  FT03_25PCNT_VALUE  "FT-3 25% Range Value For HMI Display" %
%   F29:31  FIC214_25PCNT  "FIC-21-4 25% Value (For HMI Display)" %
%   F26:130  FT03_MIN  "FT-3 Minimum Value" %
%   F29:30  FIC214_MIN  "FIC-21-4 0% Value (For HMI Display)" %
%   F26:131  FT03_MAX  "FT-3 Maximum Value" %
%   F29:34  FIC214_MAX  "FIC-21-4 100% Value (For HMI Display)" %
%   N11:223  FT03_PID_MAX  "FT-3 Flow Transmitter No-3 PID Statement Maximum Input Value" %
%   N16:37  FIC214_SMAX  "FIC-21-4 Feed Flow No-4 Setpoint Maximum" %
%   N11:213  FT03_PID_MIN  "FT-3 Flow Transmitter No-3 PID Statement Minimum Input Value" %
%   N16:38  FIC214_SMIN  "FIC-21-4 Feed Flow No-4 Setpoint Minimum" %

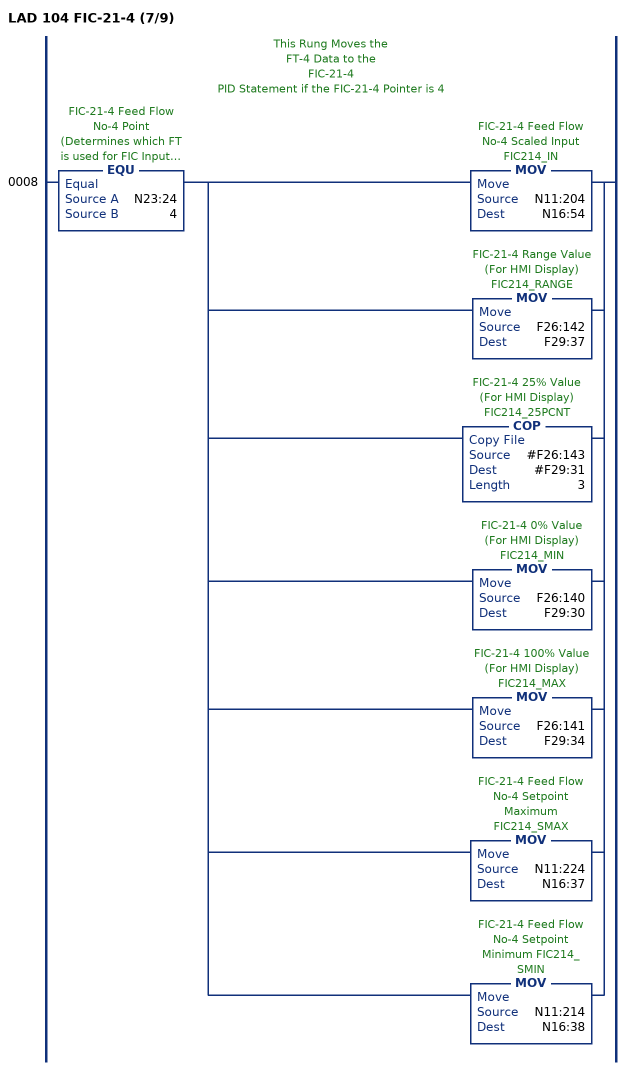
% Rung: 8 %
% This Rung Moves the
% FT-4 Data to the
% FIC-21-4
% PID Statement if the FIC-21-4 Pointer is 4 %
SOR EQU N23:24 4 BST MOV N11:204 N16:54 NXB MOV F26:142 F29:37 NXB COP #F26:143 #F29:31 3 NXB MOV F26:140 F29:30 NXB MOV F26:141 F29:34 NXB MOV N11:224 N16:37 NXB MOV N11:214 N16:38 BND EOR
%   N23:24  FIC214_IN_PTR  "FIC-21-4 Feed Flow No-4 Point (Determines which FT is used for FIC Input)" %
%   N11:204  FT04_PID_IN  "FT-4 Flow Transmitter No-4 PID Statement Input Value" %
%   N16:54  FIC214_IN  "FIC-21-4 Feed Flow No-4 Scaled Input" %
%   F26:142  FT04_RANGE  "FT-4 Range Value (Max-Min)" %
%   F29:37  FIC214_RANGE  "FIC-21-4 Range Value (For HMI Display)" %
%   F26:143  FT04_25PCNT_VALUE  "FT-4 25% Range Value For HMI Display" %
%   F29:31  FIC214_25PCNT  "FIC-21-4 25% Value (For HMI Display)" %
%   F26:140  FT04_MIN  "FT-4 Minimum Value" %
%   F29:30  FIC214_MIN  "FIC-21-4 0% Value (For HMI Display)" %
%   F26:141  FT04_MAX  "FT-4 Maximum Value" %
%   F29:34  FIC214_MAX  "FIC-21-4 100% Value (For HMI Display)" %
%   N11:224  FT04_PID_MAX  "FT-4 Flow Transmitter No-4 PID Statement Maximum Input Value" %
%   N16:37  FIC214_SMAX  "FIC-21-4 Feed Flow No-4 Setpoint Maximum" %
%   N11:214  FT04_PID_MIN  "FT-4 Flow Transmitter No-4 PID Statement Minimum Input Value" %
%   N16:38  FIC214_SMIN  "FIC-21-4 Feed Flow No-4 Setpoint Minimum" %

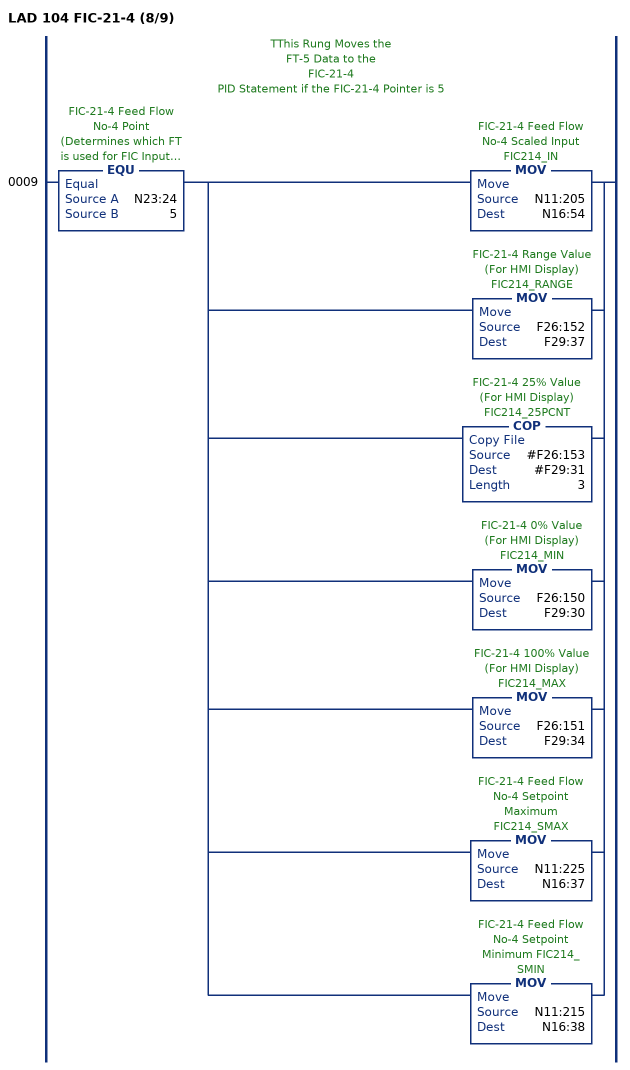
% Rung: 9 %
% TThis Rung Moves the
% FT-5 Data to the
% FIC-21-4
% PID Statement if the FIC-21-4 Pointer is 5 %
SOR EQU N23:24 5 BST MOV N11:205 N16:54 NXB MOV F26:152 F29:37 NXB COP #F26:153 #F29:31 3 NXB MOV F26:150 F29:30 NXB MOV F26:151 F29:34 NXB MOV N11:225 N16:37 NXB MOV N11:215 N16:38 BND EOR
%   N23:24  FIC214_IN_PTR  "FIC-21-4 Feed Flow No-4 Point (Determines which FT is used for FIC Input)" %
%   N11:205  FT05_PID_IN  "FT-5 Flow Transmitter No-5 PID Statement Input Value" %
%   N16:54  FIC214_IN  "FIC-21-4 Feed Flow No-4 Scaled Input" %
%   F26:152  FT05_RANGE  "FT-5 Range Value (Max-Min)" %
%   F29:37  FIC214_RANGE  "FIC-21-4 Range Value (For HMI Display)" %
%   F26:153  FT05_25PCNT_VALUE  "FT-5 25% Range Value For HMI Display" %
%   F29:31  FIC214_25PCNT  "FIC-21-4 25% Value (For HMI Display)" %
%   F26:150  FT05_MIN  "FT-5 Minimum Value" %
%   F29:30  FIC214_MIN  "FIC-21-4 0% Value (For HMI Display)" %
%   F26:151  FT05_MAX  "FT-5 Maximum Value" %
%   F29:34  FIC214_MAX  "FIC-21-4 100% Value (For HMI Display)" %
%   N11:225  FT05_PID_MAX  "FT-5 Flow Transmitter No-5 PID Statement Maximum Input Value" %
%   N16:37  FIC214_SMAX  "FIC-21-4 Feed Flow No-4 Setpoint Maximum" %
%   N11:215  FT05_PID_MIN  "FT-5 Flow Transmitter No-5 PID Statement Minimum Input Value" %
%   N16:38  FIC214_SMIN  "FIC-21-4 Feed Flow No-4 Setpoint Minimum" %

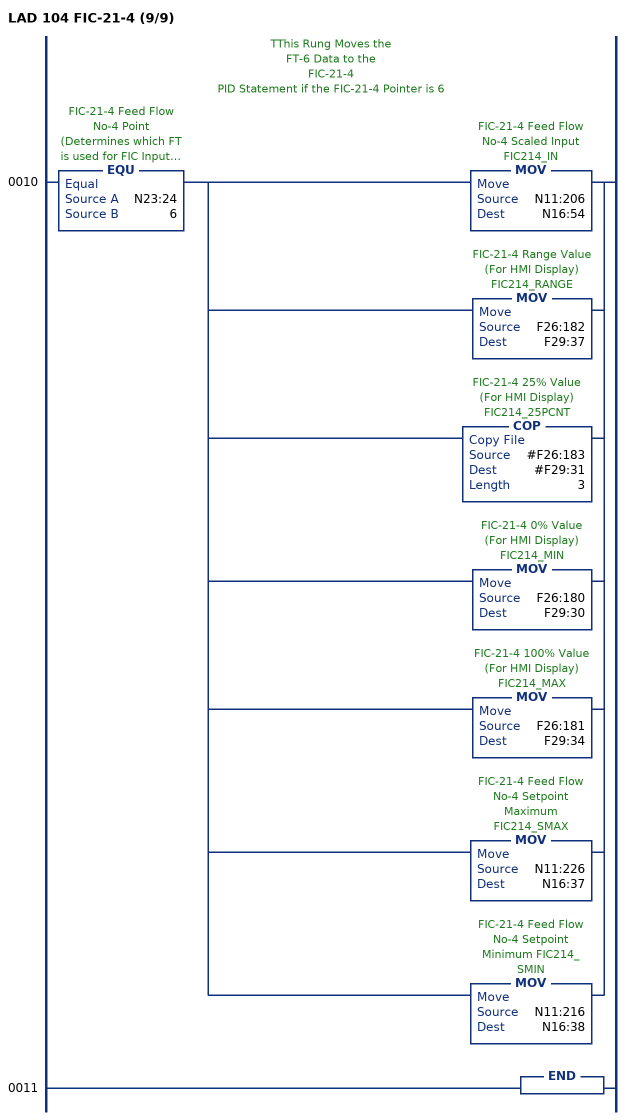
% Rung: 10 %
% TThis Rung Moves the
% FT-6 Data to the
% FIC-21-4
% PID Statement if the FIC-21-4 Pointer is 6 %
SOR EQU N23:24 6 BST MOV N11:206 N16:54 NXB MOV F26:182 F29:37 NXB COP #F26:183 #F29:31 3 NXB MOV F26:180 F29:30 NXB MOV F26:181 F29:34 NXB MOV N11:226 N16:37 NXB MOV N11:216 N16:38 BND EOR
%   N23:24  FIC214_IN_PTR  "FIC-21-4 Feed Flow No-4 Point (Determines which FT is used for FIC Input)" %
%   N11:206  FT06_PID_IN  "FT-6 Flow Transmitter No-6 PID Statement Input Value" %
%   N16:54  FIC214_IN  "FIC-21-4 Feed Flow No-4 Scaled Input" %
%   F26:182  FT06_RANGE  "FT-6 Range Value (Max-Min)" %
%   F29:37  FIC214_RANGE  "FIC-21-4 Range Value (For HMI Display)" %
%   F26:183  FT06_25PCNT_VALUE  "FT-6 25% Range Value For HMI Display" %
%   F29:31  FIC214_25PCNT  "FIC-21-4 25% Value (For HMI Display)" %
%   F26:180  FT06_MIN  "FT-6 Minimum Value" %
%   F29:30  FIC214_MIN  "FIC-21-4 0% Value (For HMI Display)" %
%   F26:181  FT06_MAX  "FT-6 Maximum Value" %
%   F29:34  FIC214_MAX  "FIC-21-4 100% Value (For HMI Display)" %
%   N11:226  FT06_PID_MAX  "FT-6 Flow Transmitter No-6 PID Statement Maximum Input Value" %
%   N16:37  FIC214_SMAX  "FIC-21-4 Feed Flow No-4 Setpoint Maximum" %
%   N11:216  FT06_PID_MIN  "FT-6 Flow Transmitter No-6 PID Statement Minimum Input Value" %
%   N16:38  FIC214_SMIN  "FIC-21-4 Feed Flow No-4 Setpoint Minimum" %
% Rung: 11 %
SOR END EOR

LADDER 111 "PIC-9-1"    % Vacuum Control No-1 PID %
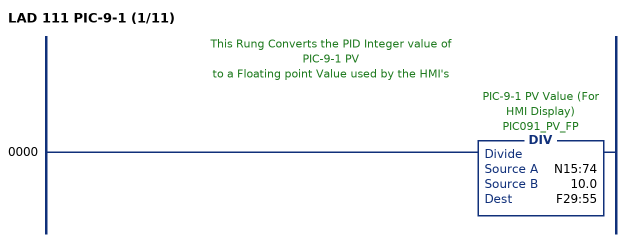
% Rung: 0 %
% This Rung Converts the PID Integer value of
% PIC-9-1 PV
% to a Floating point Value used by the HMI's %
SOR DIV N15:74 10.0 F29:55 EOR
%   N15:74  PIC091_PV  "PIC-9-1 Vacuum Press No-1 Scaled Process Variable" %
%   F29:55  PIC091_PV_FP  "PIC-9-1 PV Value (For HMI Display)" %

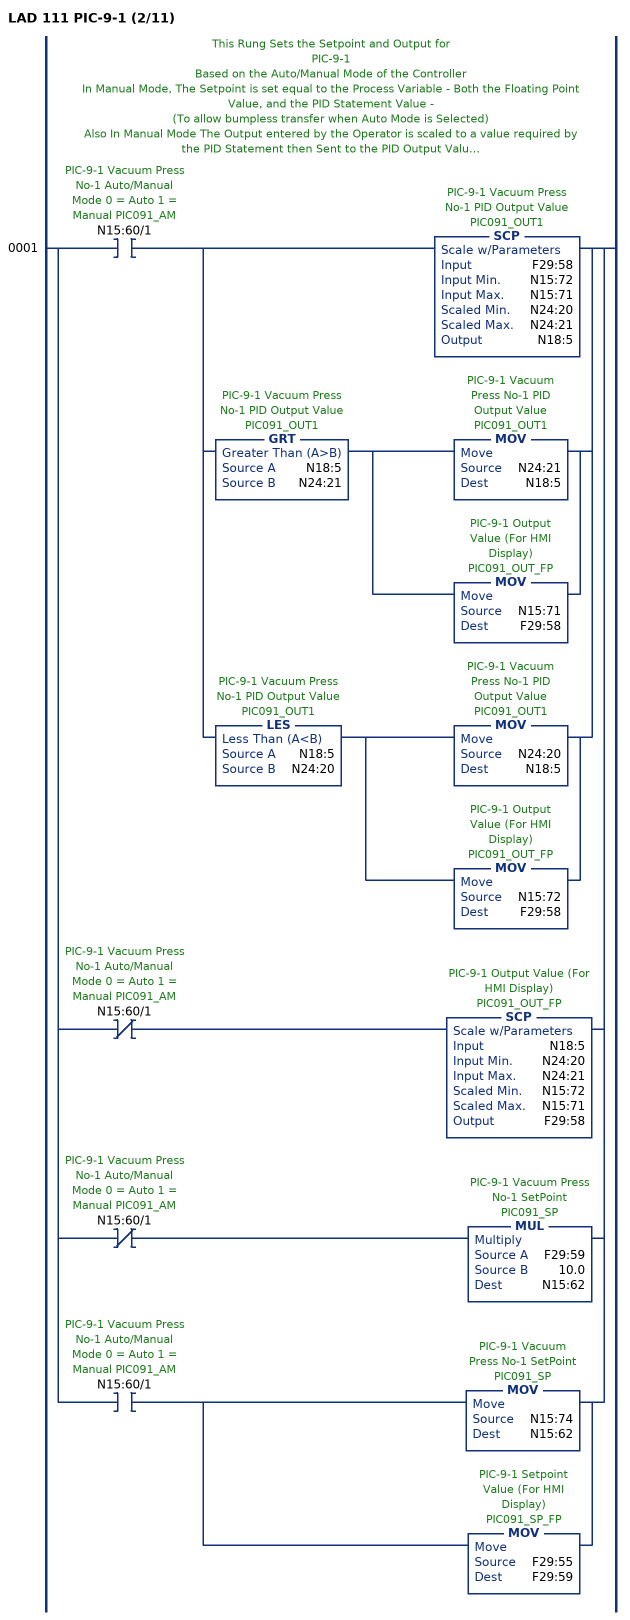
% Rung: 1 %
% This Rung Sets the Setpoint and Output for
% PIC-9-1
% Based on the Auto/Manual Mode of the Controller
% In Manual Mode, The Setpoint is set equal to the Process Variable - Both the Floating Point Value, and the PID Statement Value -
% (To allow bumpless transfer when Auto Mode is Selected)
% Also In Manual Mode The Output entered by the Operator is scaled to a value required by the PID Statement then Sent to the PID Output Value
% 
% In Auto Mode, The Setpoint is Entered by the Operator from Any HMI terminal, Multiplied by 10, and placed in the PID Statement's Setpoint Location
% Also In Auto Mode, the Output (used by the Operator) is set equal to the actual value of the pID statement
% (To allow bumpless transfer when Manual Mode is Selected) %
SOR BST XIC N15:60/1 BST SCP F29:58 N15:72 N15:71 N24:20 N24:21 N18:5 NXB GRT N18:5 N24:21 BST MOV N24:21 N18:5 NXB MOV N15:71 F29:58 BND NXB LES N18:5 N24:20 BST MOV N24:20 N18:5 NXB MOV N15:72 F29:58 BND BND NXB XIO N15:60/1 SCP N18:5 N24:20 N24:21 N15:72 N15:71 F29:58 NXB XIO N15:60/1 MUL F29:59 10.0 N15:62 NXB XIC N15:60/1 BST MOV N15:74 N15:62 NXB MOV F29:55 F29:59 BND BND EOR
%   N15:60/1  PIC091_AM  "PIC-9-1 Vacuum Press No-1 Auto/Manual Mode 0 = Auto 1 = Manual" %
%   F29:58  PIC091_OUT_FP  "PIC-9-1 Output Value (For HMI Display)" %
%   N15:72  PIC091_OMIN  "PIC-9-1 Vacuum Press No-1 Output Minimum" %
%   N15:71  PIC091_OMAX  "PIC-9-1 Vacuum Press No-1 Output Maximum" %
%   N24:20  PID_MIN  "PID Statement Minimum Value" %
%   N24:21  PID_MAX  "PID Statement Maximum Value" %
%   N18:5  PIC091_OUT1  "PIC-9-1 Vacuum Press No-1 PID Output Value" %
%   F29:59  PIC091_SP_FP  "PIC-9-1 Setpoint Value (For HMI Display)" %
%   N15:62  PIC091_SP  "PIC-9-1 Vacuum Press No-1 SetPoint" %
%   N15:74  PIC091_PV  "PIC-9-1 Vacuum Press No-1 Scaled Process Variable" %
%   F29:55  PIC091_PV_FP  "PIC-9-1 PV Value (For HMI Display)" %

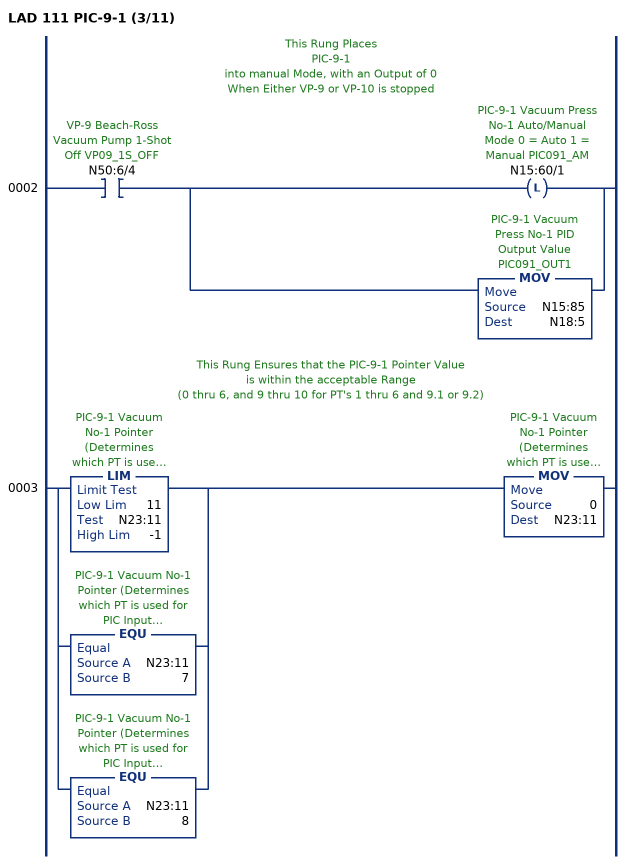
% Rung: 2 %
% This Rung Places
% PIC-9-1
% into manual Mode, with an Output of 0
% When Either VP-9 or VP-10 is stopped %
SOR XIC N50:6/4 BST OTL N15:60/1 NXB MOV N15:85 N18:5 BND EOR
%   N50:6/4  VP09_1S_OFF  "VP-9 Beach-Ross Vacuum Pump 1-Shot Off" %
%   N15:60/1  PIC091_AM  "PIC-9-1 Vacuum Press No-1 Auto/Manual Mode 0 = Auto 1 = Manual" %
%   N15:85  PIC091_OFF_OUTPUT  "PIC-9-1 Output When VP-9 and VP-10 Are Off" %
%   N18:5  PIC091_OUT1  "PIC-9-1 Vacuum Press No-1 PID Output Value" %
% Rung: 3 %
% This Rung Ensures that the PIC-9-1 Pointer Value
% is within the acceptable Range
% (0 thru 6, and 9 thru 10 for PT's 1 thru 6 and 9.1 or 9.2) %
SOR BST LIM 11 N23:11 -1 NXB EQU N23:11 7 NXB EQU N23:11 8 BND MOV 0 N23:11 EOR
%   N23:11  PIC091_IN_PTR  "PIC-9-1 Vacuum No-1 Pointer (Determines which PT is used for PIC Input)" %

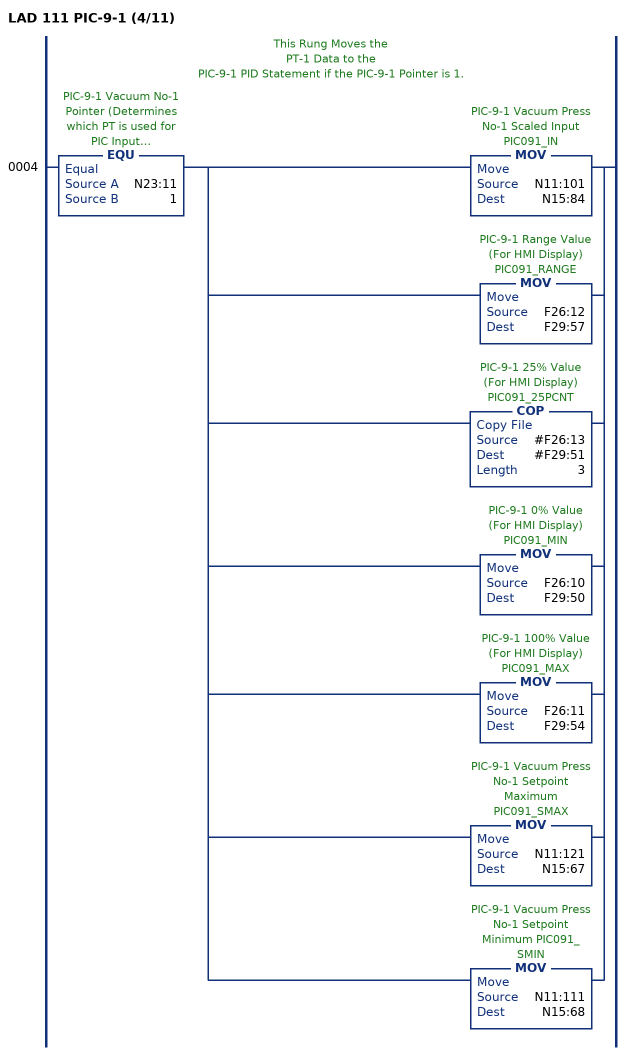
% Rung: 4 %
% This Rung Moves the
% PT-1 Data to the
% PIC-9-1 PID Statement if the PIC-9-1 Pointer is 1. %
SOR EQU N23:11 1 BST MOV N11:101 N15:84 NXB MOV F26:12 F29:57 NXB COP #F26:13 #F29:51 3 NXB MOV F26:10 F29:50 NXB MOV F26:11 F29:54 NXB MOV N11:121 N15:67 NXB MOV N11:111 N15:68 BND EOR
%   N23:11  PIC091_IN_PTR  "PIC-9-1 Vacuum No-1 Pointer (Determines which PT is used for PIC Input)" %
%   N11:101  PT01_PID_IN  "PT-01 Vacuum Transmitter No-1 PID Statement Input Value" %
%   N15:84  PIC091_IN  "PIC-9-1 Vacuum Press No-1 Scaled Input" %
%   F26:12  PT01_RANGE  "PT-1 Range Value (Max-Min)" %
%   F29:57  PIC091_RANGE  "PIC-9-1 Range Value (For HMI Display)" %
%   F26:13  PT01_25PCNT_VALUE  "PT-1 25% Range Value For HMI Display" %
%   F29:51  PIC091_25PCNT  "PIC-9-1 25% Value (For HMI Display)" %
%   F26:10  PT01_MIN  "PT-1 Minimum Value" %
%   F29:50  PIC091_MIN  "PIC-9-1 0% Value (For HMI Display)" %
%   F26:11  PT01_MAX  "PT-1 Maximum Value" %
%   F29:54  PIC091_MAX  "PIC-9-1 100% Value (For HMI Display)" %
%   N11:121  PT01_PID_MAX  "PT-01 Vacuum Transmitter No-1 PID Statement Maximum Input Value" %
%   N15:67  PIC091_SMAX  "PIC-9-1 Vacuum Press No-1 Setpoint Maximum" %
%   N11:111  PT01_PID_MIN  "PT-01 Vacuum Transmitter No-1 PID Statement Minimum Input Value" %
%   N15:68  PIC091_SMIN  "PIC-9-1 Vacuum Press No-1 Setpoint Minimum" %

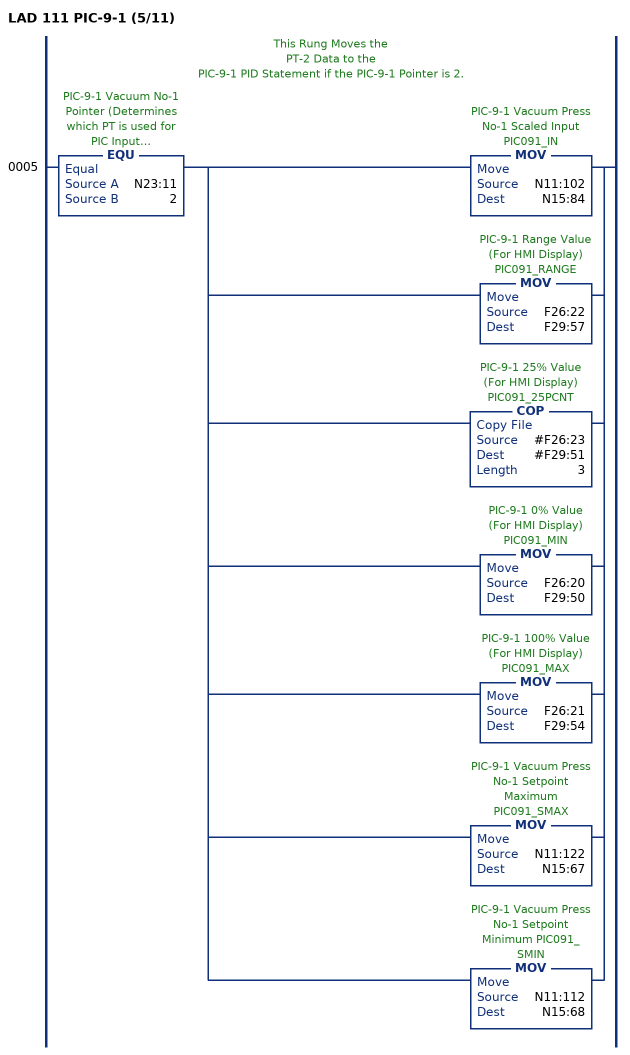
% Rung: 5 %
% This Rung Moves the
% PT-2 Data to the
% PIC-9-1 PID Statement if the PIC-9-1 Pointer is 2. %
SOR EQU N23:11 2 BST MOV N11:102 N15:84 NXB MOV F26:22 F29:57 NXB COP #F26:23 #F29:51 3 NXB MOV F26:20 F29:50 NXB MOV F26:21 F29:54 NXB MOV N11:122 N15:67 NXB MOV N11:112 N15:68 BND EOR
%   N23:11  PIC091_IN_PTR  "PIC-9-1 Vacuum No-1 Pointer (Determines which PT is used for PIC Input)" %
%   N11:102  PT02_PID_IN  "PT-02 Vacuum Transmitter No-2 PID Statement Input Value" %
%   N15:84  PIC091_IN  "PIC-9-1 Vacuum Press No-1 Scaled Input" %
%   F26:22  PT02_RANGE  "PT-2 Range Value (Max-Min)" %
%   F29:57  PIC091_RANGE  "PIC-9-1 Range Value (For HMI Display)" %
%   F26:23  PT02_25PCNT_VALUE  "PT-2 25% Range Value For HMI Display" %
%   F29:51  PIC091_25PCNT  "PIC-9-1 25% Value (For HMI Display)" %
%   F26:20  PT02_MIN  "PT-2 Minimum Value" %
%   F29:50  PIC091_MIN  "PIC-9-1 0% Value (For HMI Display)" %
%   F26:21  PT02_MAX  "PT-2 Maximum Value" %
%   F29:54  PIC091_MAX  "PIC-9-1 100% Value (For HMI Display)" %
%   N11:122  PT02_PID_MAX  "PT-02 Vacuum Transmitter No-2 PID Statement Maximum Input Value" %
%   N15:67  PIC091_SMAX  "PIC-9-1 Vacuum Press No-1 Setpoint Maximum" %
%   N11:112  PT02_PID_MIN  "PT-02 Vacuum Transmitter No-2 PID Statement Minimum Input Value" %
%   N15:68  PIC091_SMIN  "PIC-9-1 Vacuum Press No-1 Setpoint Minimum" %

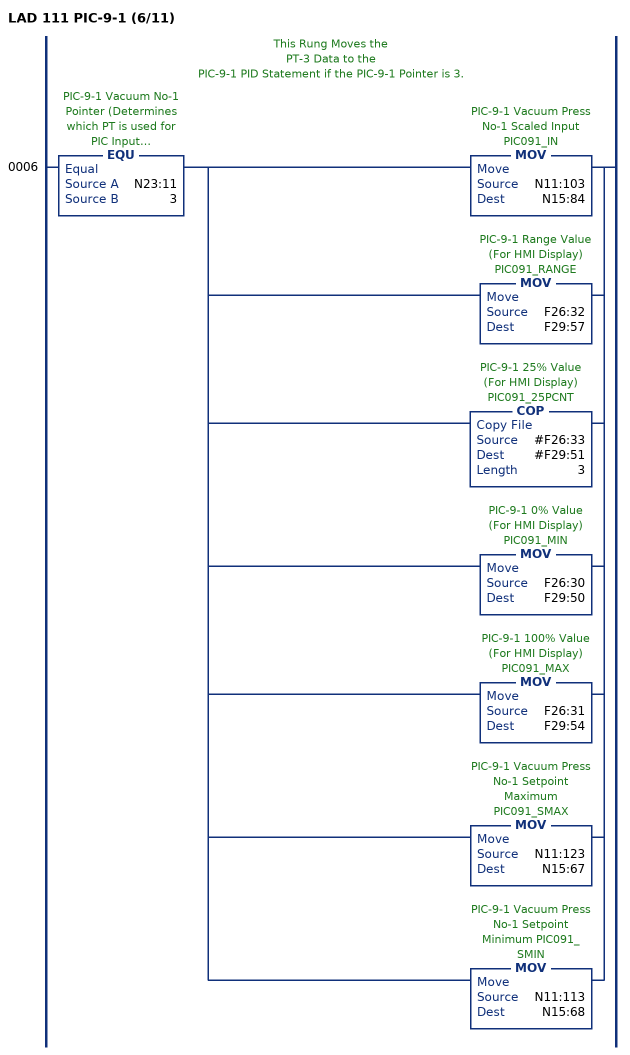
% Rung: 6 %
% This Rung Moves the
% PT-3 Data to the
% PIC-9-1 PID Statement if the PIC-9-1 Pointer is 3. %
SOR EQU N23:11 3 BST MOV N11:103 N15:84 NXB MOV F26:32 F29:57 NXB COP #F26:33 #F29:51 3 NXB MOV F26:30 F29:50 NXB MOV F26:31 F29:54 NXB MOV N11:123 N15:67 NXB MOV N11:113 N15:68 BND EOR
%   N23:11  PIC091_IN_PTR  "PIC-9-1 Vacuum No-1 Pointer (Determines which PT is used for PIC Input)" %
%   N11:103  PT03_PID_IN  "PT-03 Vacuum Transmitter No-3 PID Statement Input Value" %
%   N15:84  PIC091_IN  "PIC-9-1 Vacuum Press No-1 Scaled Input" %
%   F26:32  PT03_RANGE  "PT-3 Range Value (Max-Min)" %
%   F29:57  PIC091_RANGE  "PIC-9-1 Range Value (For HMI Display)" %
%   F26:33  PT03_25PCNT_VALUE  "PT-3 25% Range Value For HMI Display" %
%   F29:51  PIC091_25PCNT  "PIC-9-1 25% Value (For HMI Display)" %
%   F26:30  PT03_MIN  "PT-3 Minimum Value" %
%   F29:50  PIC091_MIN  "PIC-9-1 0% Value (For HMI Display)" %
%   F26:31  PT03_MAX  "PT-3 Maximum Value" %
%   F29:54  PIC091_MAX  "PIC-9-1 100% Value (For HMI Display)" %
%   N11:123  PT03_PID_MAX  "PT-03 Vacuum Transmitter No-3 PID Statement Maxmium Input Value" %
%   N15:67  PIC091_SMAX  "PIC-9-1 Vacuum Press No-1 Setpoint Maximum" %
%   N11:113  PT03_PID_MIN  "PT-03 Vacuum Transmitter No-3 PID Statement Minimum Input Value" %
%   N15:68  PIC091_SMIN  "PIC-9-1 Vacuum Press No-1 Setpoint Minimum" %

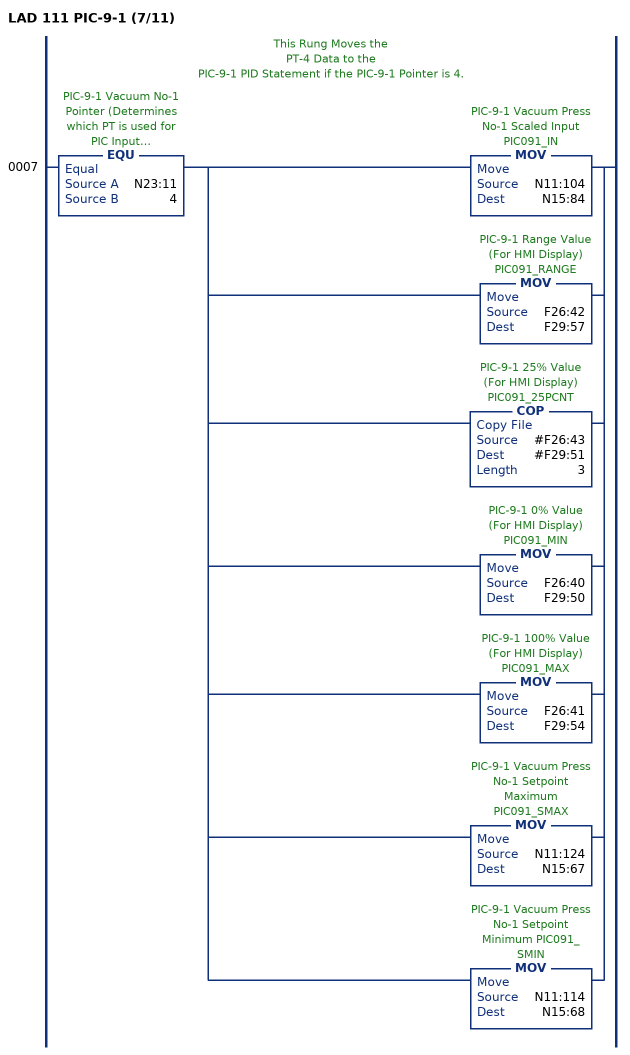
% Rung: 7 %
% This Rung Moves the
% PT-4 Data to the
% PIC-9-1 PID Statement if the PIC-9-1 Pointer is 4. %
SOR EQU N23:11 4 BST MOV N11:104 N15:84 NXB MOV F26:42 F29:57 NXB COP #F26:43 #F29:51 3 NXB MOV F26:40 F29:50 NXB MOV F26:41 F29:54 NXB MOV N11:124 N15:67 NXB MOV N11:114 N15:68 BND EOR
%   N23:11  PIC091_IN_PTR  "PIC-9-1 Vacuum No-1 Pointer (Determines which PT is used for PIC Input)" %
%   N11:104  PT04_PID_IN  "PT-04 Vacuum Transmitter No-4 PID Statement Input Value" %
%   N15:84  PIC091_IN  "PIC-9-1 Vacuum Press No-1 Scaled Input" %
%   F26:42  PT04_RANGE  "PT-4 Range Value (Max-Min)" %
%   F29:57  PIC091_RANGE  "PIC-9-1 Range Value (For HMI Display)" %
%   F26:43  PT04_25PCNT_VALUE  "PT-4 25% Range Value For HMI Display" %
%   F29:51  PIC091_25PCNT  "PIC-9-1 25% Value (For HMI Display)" %
%   F26:40  PT04_MIN  "PT-4 Minimum Value" %
%   F29:50  PIC091_MIN  "PIC-9-1 0% Value (For HMI Display)" %
%   F26:41  PT04_MAX  "PT-4 Maximum Value" %
%   F29:54  PIC091_MAX  "PIC-9-1 100% Value (For HMI Display)" %
%   N11:124  PT04_PID_MAX  "PT-04 Vacuum Transmitter No-4 PID Statement Maximum Input Value" %
%   N15:67  PIC091_SMAX  "PIC-9-1 Vacuum Press No-1 Setpoint Maximum" %
%   N11:114  PT04_PID_MIN  "PT-04 Vacuum Transmitter No-4 PID Statement Minimum Input Value" %
%   N15:68  PIC091_SMIN  "PIC-9-1 Vacuum Press No-1 Setpoint Minimum" %

